Universal Robots PolyScope program: Camera_not_on_robot_example_1.1.1.urp

Program Camera_not_on_robot_example_1.1.1 (installation=default directory=/ursim/programs createdIn=5.13.0 lastSavedIn=5.25.1 robotSerialNumber=20195599999)
Calibrated DH parameters: a=[0, -0.425, -0.3922, 0, 0, 0]; d=[0.1625, 0, 0, 0.1333, 0.0997, 0.0996]; alpha=[1.570796, 0, 0, 1.570796, -1.570796, 0]; deltaTheta=[0, 0, 0, 0, 0, 0]
InitVariablesNode variables(variable(name=we_custom_value, expression="0"), variable(name=we_logging_on, expression=False), variable(name=we_num_objects, expression=0), variable(name=we_object_pose, expression=p[0.0,0.0,0.0,0.0,0.0,0.0]), variable(name=we_pose_valid, expression=False), variable(name=we_shape_model, expression=0), variable(name=we_target_pose, expression=p[0.0,0.0,0.0,0.0,0.0,0.0]))
BeforeStart
  poses_taught := False
Robot Program (runOnlyOnce=true)
  Call single_detection
SubProgram -> single_detection
SubProgram multi_detection (keepSynchronizedWithDisk=false)
  URCap Change job (wenglor robotVision, wenglor sensoric elektronische Geräte GmbH) dataModel(jobNameKey=find_objects.u3p, Variable(key=we_logging_onKey, variable=we_logging_on))
  MoveJ speed 60 deg/s, acceleration 80 deg/s^2 (useActiveTCP=true optimoveEnabled=false optiMoveSpeed=0.3 optiMoveAcceleration=0.09) feature=Base
    Waypoint detection_pose: 
  URCap Detect objects (wenglor robotVision, wenglor sensoric elektronische Geräte GmbH) dataModel(Variable(key=we_num_objectsKey, variable(name=we_num_objects, initializeExpression=0)), Variable(key=we_logging_onKey, variable=we_logging_on))
    Loop While (checkContinuously=false) expression=we_num_objects > 0
      URCap Get object pose (wenglor robotVision, wenglor sensoric elektronische Geräte GmbH) dataModel(Variable(key=we_object_poseKey, variable=we_object_pose), Variable(key=we_shape_modelKey, variable=we_shape_model), Variable(key=we_custom_valueKey, variable=we_custom_value), Variable(key=we_pose_validKey, variable=we_pose_valid))
        If we_pose_valid == False
          'Add error handling here'
          Popup Error (haltProgram=false message=Pose not valid. inputType=Text)
          Halt
        If is_within_safety_limits(we_object_pose) == False
          'Add error handling here'
          Popup Error (haltProgram=false message=Pose cannot be reached by the robot. inputType=Text)
          Halt
        'Movement and gripping here'
        'Add conditional checks for we_shape_model for we_custom_value'
        Folder Pick object
          'Move to object with reduced speed'
          MoveL speed 90 mm/s, acceleration 400 mm/s^2 (useActiveTCP=true optimoveEnabled=false optiMoveSpeed=0.3 optiMoveAcceleration=0.09) feature=Base
            Waypoint Variable (Variable): variable=we_object_pose
          'Placeholder - Grip object'
        Folder Place object
          'Placeholder - Move to place pose'
          'Placeholder - Drop object'
      'Necessary to prevent index errors'
      we_num_objects := we_num_objects - 1
SubProgram update_reference_frame (keepSynchronizedWithDisk=false)
  URCap Change job (wenglor robotVision, wenglor sensoric elektronische Geräte GmbH) dataModel(jobNameKey=find_target.u3p)
  'Move to pose where target is visible'
  MoveJ speed 60 deg/s, acceleration 80 deg/s^2 (useActiveTCP=true optimoveEnabled=false optiMoveSpeed=0.3 optiMoveAcceleration=0.09) feature=Base
    Waypoint target_detect_p: 
  URCap Detect target (wenglor robotVision, wenglor sensoric elektronische Geräte GmbH) dataModel(targetSelectorDetectTargetIndexKey=0, Variable(key=we_target_poseKey, variable(name=we_target_pose, initializeExpression=p[0.0,0.0,0.0,0.0,0.0,0.0])), Variable(key=we_custom_valueKey, variable=we_custom_value), Variable(key=we_pose_validKey, variable=we_pose_valid))
    If we_pose_valid == False
      'Add error handling here'
      Popup Error (haltProgram=false message=Pose not valid. inputType=Text)
      Halt
    If is_within_safety_limits(we_target_pose) == False
      'Add error handling here'
      Popup Error (haltProgram=false message=Pose cannot be reached by the robot. inputType=Text)
      Halt
  w_ref_frame := we_target_pose
  If poses_taught == False
    Popup Message (haltProgram=false message='Reference frame updated. Please update poses now relative to w_ref_frame' inputType=Text)
    Popup Message (haltProgram=false message='Set poses_taught to True and restart the program after teaching the poses. inputType=Text)
    Halt
  'The machine reference frame is now updated, and so are the poses inside the machine.'
  'Move to poses in the machine that were taught relative to `w_reference_frame`.'
  MoveL speed 250 mm/s, acceleration 1200 mm/s^2 (useActiveTCP=true optimoveEnabled=false optiMoveSpeed=0.3 optiMoveAcceleration=0.09) feature=w_ref_frame
    Waypoint pose_in_machine: 
SubProgram single_detection (keepSynchronizedWithDisk=false)
  URCap Change job (wenglor robotVision, wenglor sensoric elektronische Geräte GmbH) dataModel(jobNameKey=find_objects.u3p, Variable(key=we_logging_onKey, variable(name=we_logging_on description=Shall wenglor nodes write messages to the robot log? - boolean type, initializeExpression=False)))
  MoveJ speed 60 deg/s, acceleration 80 deg/s^2 (useActiveTCP=true optimoveEnabled=false optiMoveSpeed=0.3 optiMoveAcceleration=0.09) feature=Base
    Waypoint detection_pose: 
  URCap Detect objects (wenglor robotVision, wenglor sensoric elektronische Geräte GmbH) dataModel(Variable(key=we_num_objectsKey, variable(name=we_num_objects, initializeExpression=0)), Variable(key=we_logging_onKey, variable=we_logging_on))
    URCap Get object pose (wenglor robotVision, wenglor sensoric elektronische Geräte GmbH) dataModel(Variable(key=we_object_poseKey, variable(name=we_object_pose description=The 3D object pose - pose type, initializeExpression=p[0.0,0.0,0.0,0.0,0.0,0.0])), Variable(key=we_shape_modelKey, variable(name=we_shape_model description=The shape model ID of the current object - integer type, initializeExpression=0)), Variable(key=we_custom_valueKey, variable(name=we_custom_value description=Can be any value linked in uniVision. In this case it is the detection score for the object. - string type, initializeExpression="0")), Variable(key=we_pose_validKey, variable(name=we_pose_valid, initializeExpression=False)))
      If we_pose_valid == False
        'Add error handling here'
        Popup Error (haltProgram=false message=Pose not valid. inputType=Text)
        Halt
      If is_within_safety_limits(we_object_pose) == False
        'Add error handling here'
        Popup Error (haltProgram=false message=Pose cannot be reached by the robot. inputType=Text)
        Halt
      'Movement and gripping here'
      'Add conditional checks for we_shape_model for we_custom_value'
      Folder Pick object
        'Move to object with reduced speed'
        MoveL speed 90 mm/s, acceleration 400 mm/s^2 (useActiveTCP=true optimoveEnabled=false optiMoveSpeed=0.3 optiMoveAcceleration=0.09) feature=Base
          Waypoint Variable (Variable): variable=we_object_pose
        'Placeholder - Grip object'
      Folder Place object
        'Placeholder - Move to place pose'
        'Placeholder - Drop object'
